{attribute 'pack_mode' := '2'}
TYPE ST_XPU_STATE :
STRUCT
  Init            : E_XPU_INIT;
  State           : E_XPU_STATE;
  Check           : E_XPU_CHECK;
  DcLink          : BIT;
END_STRUCT
END_TYPE

(* stored: Version 1.1.0.1, ProductVersion 3.1.4024.12
   DUT ST_XPU_STATE: Id {bd870dc8-c733-43d8-82f8-72ebd203def0} *)
